INTERFACE ITF_ITC_Emulation EXTENDS __System.IQueryInterface

METHOD M_AddData : BOOL
VAR_INPUT
	meChannelSrc	: E_MFCS_Channel;
	mMsgType		: INT;
	mpData			: PVOID;
	mLen			: UDINT;
END_VAR
END_METHOD

METHOD M_CallITC_Service : BOOL
VAR_INPUT
END_VAR
END_METHOD

END_INTERFACE

(* stored: Version 1.1.0.1, ProductVersion 3.1.4022.12
   Itf ITF_ITC_Emulation: Id {c08ae787-d516-43b7-b6e7-01e8d23f907e}
   Method M_AddData: Id {e4491b33-db3d-4fa9-a0bb-3814ac9c7ec8}
   Method M_CallITC_Service: Id {35d5f416-1a65-4131-a715-2f691f09f57e} *)
